{attribute 'object_name' := 'sta_TurnEmptyBusy'}
METHOD PROTECTED sta_TurnEmptyBusy : BOOL
// state implemetation
//--------------------------------------------------------------------------------------
// Entry action
	IF (me.StateMachine.intState<>me.StateMachine.intStateLastCycle) THEN
		me.StateMachine.intStateLastCycle := me.StateMachine.intState;
//		Log Message ---------------------
//		TC2_SYSTEM.ADSLOGSTR(ADSLOG_MSGTYPE_LOG,'%s','sta_TurnEmptyBusy');
//		---------------------------------
		(*p_fbMalteser^.CtrlSIf^.Par.*)intTurnDirection := E_TURN_DIRECTION.AUTOMATIC;
		(*p_fbMalteser^.CtrlSIf^.Par.*)uinPositionToGo := SIf.Cur.rInOutPosition.uinInput;
		
		IF (SIf.Cfg.bolRaxEnable) THEN
			IF SIf.Cur.rInOutPosition.uinInput*90*10 = p_fbRAX^.CtrlSIf^.Cur.dinModPosition_0_1deg THEN
				p_fbRAX^.CtrlCIf^.Job.intACmd := cCMD_STOP;
				me.SubStateMachine.intState := PTS_CmdState.cSUB_WAIT_DONE;
				me.SubStateMachine.intStateNext := PTS_CmdState.cSUB_WAIT_DONE;
			ELSE	
				p_fbRAX^.CtrlCIf^.Job.intACmd := RAX_CmdState.cCMD_TURN;
				me.SubStateMachine.intState := PTS_CmdState.cSUB_TURNbusy;
				me.SubStateMachine.intStateNext := PTS_CmdState.cSUB_TURNbusy;
			END_IF
		ELSE
			IF SIf.Cur.rInOutPosition.uinInput = p_fbMalteser^.CtrlSIf^.Cur.uintActualPosition THEN
				p_fbMalteser^.CtrlCIf^.Job.intACmd := BASE_PLC.cCMD_RUN;
				me.SubStateMachine.intState := PTS_CmdState.cSUB_WAIT_DONE;
				me.SubStateMachine.intStateNext := PTS_CmdState.cSUB_WAIT_DONE;
			ELSE	
				p_fbMalteser^.CtrlCIf^.Job.intACmd := MDC_CmdState.cCMD_TURN;
				me.SubStateMachine.intState := PTS_CmdState.cSUB_TURNbusy;
				me.SubStateMachine.intStateNext := PTS_CmdState.cSUB_TURNbusy;
			END_IF
		END_IF
	END_IF


//--------------------------------------------------------------------------------------
// Cyclic action
	IF (me.StateMachine.intState=me.StateMachine.intStateLastCycle) THEN
		//--------------------------------------------------------------------------------------
		// sub state machine for sequence
		IF (SIf.Cfg.bolRaxEnable) THEN
			CASE me.SubStateMachine.intState OF
				//--------------------------------------------------------------------------------------
				PTS_CmdState.cSUB_TURNbusy :
					IF (p_fbRAX^.CtrlCIf^.Job.intState = RAX_CmdState.cSTA_TURN) THEN
						p_fbRAX^.CtrlCIf^.Job.intACmd := cCMD_STOP;
						me.SubStateMachine.intStateNext := PTS_CmdState.cSUB_WAIT_DONE;
					END_IF
				//--------------------------------------------------------------------------------------
				PTS_CmdState.cSUB_WAIT_DONE:
					IF (p_fbRAX^.CtrlCIf^.Job.intState = cSTA_STOP) THEN
						IF SIf.Par.eMode = E_PTS_MODE.Distribute THEN
							SIf.Cur.iActualDistributionIndex := (SIf.Cur.iActualDistributionIndex + 1) MOD PTS_CmdState.cPTS_MAX_DISTRIBUTION;	
						END_IF
	
						me.StateMachine.intStateNext := BASE_PLC.cSTA_RUNBusy;
					END_IF
				//--------------------------------------------------------------------------------------
			END_CASE
		ELSE			
			CASE me.SubStateMachine.intState OF
				//--------------------------------------------------------------------------------------
				PTS_CmdState.cSUB_TURNbusy :
					IF (p_fbMalteser^.CtrlCIf^.Job.intState = MDC_CmdState.cSTA_TURNDONE) THEN
						p_fbMalteser^.CtrlCIf^.Job.intACmd := BASE_PLC.cCMD_RUN;
						me.SubStateMachine.intStateNext := PTS_CmdState.cSUB_WAIT_DONE;
					END_IF
				//--------------------------------------------------------------------------------------
				PTS_CmdState.cSUB_WAIT_DONE:
					IF (p_fbMalteser^.CtrlCIf^.Job.intState = MDC_CmdState.cSTA_InPosition) THEN
						IF SIf.Par.eMode = E_PTS_MODE.Distribute THEN
							SIf.Cur.iActualDistributionIndex := (SIf.Cur.iActualDistributionIndex + 1) MOD PTS_CmdState.cPTS_MAX_DISTRIBUTION;	
						END_IF
	
						me.StateMachine.intStateNext := BASE_PLC.cSTA_RUNBusy;
					END_IF
				//--------------------------------------------------------------------------------------
			END_CASE
		END_IF
	END_IF


//--------------------------------------------------------------------------------------
// Exit action
	IF (me.StateMachine.intState<>me.StateMachine.intStateNext) THEN
		;
	END_IF
END_METHOD

{attribute 'object_name' := 'IoOutBridge'}
METHOD PROTECTED IoOutBridge : BOOL
VAR
	bolSwitchValvesOff: BOOL;
END_VAR
// digitale and analoge inputs read from hardware or forcing
IF (CIf.SwCfg.bolSimulation = FALSE) THEN
	;
END_IF

// Write Outputs to Turning Child (Malteser or ServoDrive)
IF (SIf.Cfg.bolRaxEnable) THEN
	// ToDo: p_fbRAX^.CtrlSIf^.Par. intTurnDirection := intTurnDirection;
	p_fbRAX^.CtrlSIf^.Par.dinPos_0_1Deg := uinPositionToGo*90*10;	
ELSE
	p_fbMalteser^.CtrlSIf^.Par.intTurnDirection := intTurnDirection;	// <0 = Turn left; =0 automatic; >0 turn right
	p_fbMalteser^.CtrlSIf^.Par.uinPositionToGo := uinPositionToGo;
END_IF
END_METHOD

{attribute 'object_name' := 'sta_PON'}
METHOD PROTECTED sta_PON : BOOL
// state implemetation
//--------------------------------------------------------------------------------------
// Entry action
	IF (me.StateMachine.intState<>me.StateMachine.intStateLastCycle) THEN
		me.StateMachine.intStateLastCycle := me.StateMachine.intState;
		
	END_IF


//--------------------------------------------------------------------------------------
// Cyclic action
	IF (me.StateMachine.intState=me.StateMachine.intStateLastCycle) THEN
		;
	END_IF




//--------------------------------------------------------------------------------------
// Exit action
	IF (me.StateMachine.intState<>me.StateMachine.intStateNext) THEN
		;
	END_IF
END_METHOD

{attribute 'object_name' := 'sta_PaperDelayBusy'}
METHOD PROTECTED sta_PaperDelayBusy : BOOL
// state implemetation
//--------------------------------------------------------------------------------------
// Entry action
	IF (me.StateMachine.intState<>me.StateMachine.intStateLastCycle) THEN
		me.StateMachine.intStateLastCycle := me.StateMachine.intState;
//		Log Message ---------------------
		TC2_SYSTEM.ADSLOGSTR(ADSLOG_MSGTYPE_LOG,'%s','sta_PaperDelayBusy');
//		---------------------------------
	END_IF


//--------------------------------------------------------------------------------------
// Cyclic action
	IF (me.StateMachine.intState = me.StateMachine.intStateLastCycle) THEN
		IF (me.StateMachine.udiTimeInState_ms > SIf.Par.udiPaperInTurnDelayTime) THEN
			me.StateMachine.intStateNext := PTS_CmdState.cSTA_TurnPaperBusy;
		END_IF
	END_IF


//--------------------------------------------------------------------------------------
// Exit action
	IF (me.StateMachine.intState<>me.StateMachine.intStateNext) THEN
		;
	END_IF
END_METHOD

{attribute 'object_name' := 'sta_RUNBusy'}
METHOD PROTECTED sta_RUNBusy : BOOL
// state implemetation
//--------------------------------------------------------------------------------------
// Entry action
IF (me.StateMachine.intState<>me.StateMachine.intStateLastCycle) THEN
	me.StateMachine.intStateLastCycle := me.StateMachine.intState;

	CASE SIf.Par.eMode OF
		E_PTS_MODE.Automatic:
			pfbAlarmCtrl^.setAlarm(CIf.Info.intCtrlId,INT_TO_UINT(E_ALM_PTS.ModeParameter),0,ADR(SIf.Alm),E_AlmState.RST,CIf.Job.eMe_ActivAlmClass);
(*
			IF SIf.Cfg.bolBarcodeReaderAvailable (* AND BCR has a new barcode read *) THEN
				me.StateMachine.intStateNext := PTS_CmdState.cSTA_GetItemBusy;
			ELSE
				pfbAlarmCtrl^.setAlarm(CIf.Info.intCtrlId,INT_TO_UINT(E_ALM_PTS.ModeParameter),0,ADR(SIf.Alm),E_AlmState.RST,CIf.Job.eMe_ActivAlmClass);
			END_IF
*)
		E_PTS_MODE.Distribute:
			SIf.Cur.rInOutPosition := SIf.Cfg.aFixPosDef[SIf.Cfg.aDistributionPositionDefinition[SIf.Cur.iActualDistributionIndex]];

		ELSE
			SIf.Cur.rInOutPosition := SIf.Cfg.aFixPosDef[SIf.Par.eMode];
	END_CASE

	(*p_fbMalteser^.CtrlSIf^.Par.*)intTurnDirection := E_TURN_DIRECTION.AUTOMATIC;
	(*p_fbMalteser^.CtrlSIf^.Par.*)uinPositionToGo := SIf.Cur.rInOutPosition.uinOutput;

	IF (SIf.Cfg.bolRaxEnable = FALSE) THEN
		IF SIf.Cfg.bolPositionMalteserEnable THEN
			p_fbMalteser^.CtrlCIf^.Job.intACmd := MDC_CmdState.cCMD_PREPOSITION;
	
			me.SubStateMachine.intState := PTS_CmdState.cSUB_PREPOSITIONbusy;
			me.SubStateMachine.intStateNext := PTS_CmdState.cSUB_PREPOSITIONbusy;
		ELSE	
			p_fbMalteser^.CtrlCIf^.Job.intACmd := BASE_PLC.cCMD_RUN;
	
			me.SubStateMachine.intState := PTS_CmdState.cSUB_WAIT_DONE;
			me.SubStateMachine.intStateNext := PTS_CmdState.cSUB_WAIT_DONE;
		END_IF
	END_IF
	
	p_fbBelt^.CtrlSIf^.Par.intDirection := E_BELT_DIRECTION.FORWARD;
	pBeltCIf^.Job.intACmd := BASE_PLC.cCMD_RUN;
END_IF


//--------------------------------------------------------------------------------------
// Cyclic action
IF (me.StateMachine.intState=me.StateMachine.intStateLastCycle) THEN

	IF (SIf.Cfg.bolRaxEnable) THEN
		me.StateMachine.intStateNext := cSTA_RUN;
	ELSE
		//--------------------------------------------------------------------------------------
		// sub state machine for sequence
		CASE me.SubStateMachine.intState OF
			//--------------------------------------------------------------------------------------
			PTS_CmdState.cSUB_PREPOSITIONbusy:
				IF (p_fbMalteser^.CtrlCIf^.Job.intState = MDC_CmdState.cSTA_PREPOSITION) THEN
					p_fbMalteser^.CtrlCIf^.Job.intACmd := BASE_PLC.cCMD_RUN;
					me.SubStateMachine.intStateNext := PTS_CmdState.cSUB_WAIT_DONE;
				END_IF
			//--------------------------------------------------------------------------------------
			PTS_CmdState.cSUB_WAIT_DONE:
				IF (p_fbMalteser^.CtrlCIf^.Job.intState = MDC_CmdState.cSTA_InPosition) 
				  AND (pBeltCIf^.Job.intState = BASE_PLC.cSTA_RUN) THEN
		//			SIf.Cur.udiPaperInTurnDelayTime := 150000 / p_fbBelt^.CtrlSIf^.Par.uinBeltSpeed;
		//			SIf.Cur.udiPaperOutTurnDelayTime := CalculateOutputDelay(p_fbBelt^.CtrlSIf^.Par.uinBeltSpeed,SIf.Cur.udiPaperInTurnDelayTime);
					me.StateMachine.intStateNext := BASE_PLC.cSTA_RUN;
				END_IF
			//--------------------------------------------------------------------------------------
		END_CASE
	END_IF
	
	IF SIf.In.bolPaperAvailable.intern THEN
		me.StateMachine.intStateNext := PTS_CmdState.cSTA_WaitPaper;
	END_IF
END_IF


//--------------------------------------------------------------------------------------
// Exit action
IF (me.StateMachine.intState<>me.StateMachine.intStateNext) THEN
	;
END_IF
END_METHOD

{attribute 'object_name' := 'sta_GetItemBusy'}
METHOD PROTECTED sta_GetItemBusy : BOOL
END_METHOD

{attribute 'object_name' := 'CtrlInit'}
METHOD CtrlInit : BOOL
SUPER^.CtrlInit();

IF (SIf.Cfg.bolRaxEnable) THEN
	THIS^.AddChild(p_fbRAX^);

	pRaxCIf := p_fbRAX^.CtrlCIf;
ELSE
	THIS^.AddChild(p_fbMalteser^);

	pMalteserCIf := p_fbMalteser^.CtrlCIf;
END_IF

THIS^.AddChild(p_fbBelt^);

pBeltCIf := p_fbBelt^.CtrlCIf;

(*
// set parent id
pMalteserCIf^.Info.intParentCtrlId := CIf.Info.intCtrlId;			
pBeltCIf^.Info.intParentCtrlId := CIf.Info.intCtrlId;			

//necessary???
THIS^.CIf.Info.p_aCIf[0] := pMalteserCIf;
THIS^.CIf.Info.p_aCIf[1] := pBeltCIf;
*)
END_METHOD

{attribute 'object_name' := 'sta_ERROR'}
METHOD PROTECTED sta_ERROR : BOOL
// state implemetation
//--------------------------------------------------------------------------------------
// Entry action
	IF (me.StateMachine.intState<>me.StateMachine.intStateLastCycle) THEN
		me.StateMachine.intStateHistory := me.StateMachine.intStateLastCycle; // -> possibillity to go back to state before error
		me.StateMachine.intStateLastCycle := me.StateMachine.intState;
		
		// stop child controllers
		pBeltCIf^.Job.intACmd := BASE_PLC.cCMD_OFF;
		IF (SIf.Cfg.bolRaxEnable) THEN
			pRaxCIf^.Job.intACmd := cCMD_OFF;
		ELSE
			pMalteserCIf^.Job.intACmd := BASE_PLC.cCMD_OFF;
		END_IF
	END_IF


//--------------------------------------------------------------------------------------
// Cyclic action
	IF (me.StateMachine.intState=me.StateMachine.intStateLastCycle) THEN
		
		;
		
		
		// State Change Condition
		IF (CIf.Job.bolAlmReset = TRUE) THEN
			me.StateMachine.intStateNext := cSTA_ERRORQuit;
		END_IF
	END_IF




//--------------------------------------------------------------------------------------
// Exit action
	IF (me.StateMachine.intState<>me.StateMachine.intStateNext) THEN
		;
	END_IF
END_METHOD

{attribute 'object_name' := 'getCtrlSIf'}
METHOD getCtrlSIf : POINTER TO T_Ctrl_SIf_PTS
getCtrlSIf := ADR(SIf);
END_METHOD

END_FUNCTION_BLOCK

// ---- POUs/Controller/Lvl2/PTS [Paper Turning Station]/helper/cycle_Pts.TcPOU
FUNCTION cycle_Pts : BOOL
VAR_INPUT
	pPts: POINTER TO T_PTS;
END_VAR

pPts^.ctrl.fbPts_Ptb_Umc.In_uinStatus 				:= pPts^.io.In_uinPtb_Umc_Status;
pPts^.ctrl.fbPts_Ptb_Umc.In_intMotorActualSpeed		:= pPts^.io.In_uinPtb_Umc_ActualSpeed;
pPts^.ctrl.fbPts_Ptb_Umc.In_uinMotorSetSpeed		:= pPts^.io.In_uinPtb_Umc_SetSpeed;
pPts^.ctrl.fbPts_Ptb_Umc.In_uinIOData				:= pPts^.io.In_uinPtb_Umc_IOData1;
pPts^.ctrl.fbPts_Ptb_Umc.In_uinECATState 			:= pPts^.io.In_uinPtb_Umc_ECatState;
pPts^.ctrl.fbPts_Ptb_Umc.In_strNetId 				:= pPts^.io.In_strPtb_Umc_ECatNetId;
pPts^.ctrl.fbPts_Ptb_Umc.In_uintPort 				:= pPts^.io.In_uinPtb_Umc_ECatPort;
pPts^.ctrl.fbPts_Ptb_Umc();
pPts^.io.Out_uinPtb_Umc_SetSpeed 					:= pPts^.ctrl.fbPts_Ptb_Umc.Out_uinSpeedSetpoint;
pPts^.io.Out_uinPtb_Umc_Control 					:= pPts^.ctrl.fbPts_Ptb_Umc.Out_uinControl;

pPts^.ctrl.fbPts_Ptb_Vpc.In_bolPumpOk 				:= pPts^.io.In_bolPtb_Vpc_PumpOk;
pPts^.ctrl.fbPts_Ptb_Vpc.In_bolVacuumOk 			:= pPts^.io.In_bolPtb_Vpc_VacuumSensor;
pPts^.ctrl.fbPts_Ptb_Vpc();
pPts^.io.Out_bolPtb_Vpc_PumpOn 						:= pPts^.ctrl.fbPts_Ptb_Vpc.Out_bolVaccumPumpOn;

IF (pPts^.ctrl.fbPts.CtrlSIf^.Cfg.bolRaxEnable = FALSE) THEN
	pPts^.ctrl.fbPts_Mdc_Umc.In_uinStatus 				:= pPts^.io.In_uinMdc_Umc_Status;
	pPts^.ctrl.fbPts_Mdc_Umc.In_intMotorActualSpeed		:= pPts^.io.In_uinMdc_Umc_ActualSpeed;
	pPts^.ctrl.fbPts_Mdc_Umc.In_uinMotorSetSpeed 		:= pPts^.io.In_uinMdc_Umc_SetSpeed;
	pPts^.ctrl.fbPts_Mdc_Umc.In_uinIOData				:= pPts^.io.In_uinMdc_Umc_IOData1;
	pPts^.ctrl.fbPts_Mdc_Umc.In_uinECATState 			:= pPts^.io.In_uinMdc_Umc_ECatState;
	pPts^.ctrl.fbPts_Mdc_Umc.In_strNetId 				:= pPts^.io.In_strMdc_Umc_ECatNetId;
	pPts^.ctrl.fbPts_Mdc_Umc.In_uintPort 				:= pPts^.io.In_uinMdc_Umc_ECatPort;
	pPts^.ctrl.fbPts_Mdc_Umc();
	pPts^.io.Out_uinMdc_Umc_SetSpeed 					:= pPts^.ctrl.fbPts_Mdc_Umc.Out_uinSpeedSetpoint;
	pPts^.io.Out_uinMdc_Umc_Control 					:= pPts^.ctrl.fbPts_Mdc_Umc.Out_uinControl;
	
	pPts^.ctrl.fbPts_Mdc.In_bolCrossPositionSensor 		:= pPts^.io.In_bolMdc_CrossPositionSensor;
	pPts^.ctrl.fbPts_Mdc.In_bolTablePositionSensor 		:= pPts^.io.In_bolMdc_TablePositionSensor;
	pPts^.ctrl.fbPts_Mdc();
ELSE
	pPts^.ctrl.fbPts_RAX_POD.In_bolHomeSwitch			:= pPts^.io.In_bolRax_PositionSensor;
	pPts^.ctrl.fbPts_RAX_POD();

	pPts^.ctrl.fbPts_RAX();
END_IF

pPts^.ctrl.fbPts_Ptb();

pPts^.ctrl.fbPts.In_bol_PaperAvailable 				:= pPts^.io.In_bolPaperSensor;
pPts^.ctrl.fbPts();

END_FUNCTION

// ---- POUs/Controller/Lvl2/PTS [Paper Turning Station]/helper/init_Pts.TcPOU
FUNCTION init_Pts : BOOL
VAR_INPUT
	pPts			: POINTER TO T_PTS;
	/// instance array of all controller instances
	pCtrlInst		: POINTER TO fb_CtrlBase;
	/// common interface array of all controllers (main use for PLC)
	pCtrlCIf		: POINTER TO T_Ctrl_CIf;
END_VAR

pPts^.ctrl.fbPts_Ptb_Vpc.iniAllCtrlArrays(pCtrlInst,pCtrlCIf,pPts^.id.Pts_Ptb_Vpc);
pPts^.ctrl.fbPts_Ptb_Umc.iniAllCtrlArrays(pCtrlInst,pCtrlCIf,pPts^.id.Pts_Ptb_Umc);
pPts^.ctrl.fbPts_Ptb.iniAllCtrlArrays(pCtrlInst,pCtrlCIf,pPts^.id.Pts_Ptb);
pPts^.ctrl.fbPts_Ptb.Drive := ADR(pPts^.ctrl.fbPts_Ptb_Umc);
pPts^.ctrl.fbPts_Ptb.VacuumPump := ADR(pPts^.ctrl.fbPts_Ptb_Vpc);

pPts^.ctrl.fbPts_Mdc_Umc.iniAllCtrlArrays(pCtrlInst,pCtrlCIf,pPts^.id.Pts_Mdc_Umc);
pPts^.ctrl.fbPts_Mdc.iniAllCtrlArrays(pCtrlInst,pCtrlCIf,pPts^.id.Pts_Mdc);
pPts^.ctrl.fbPts_Mdc.Drive := ADR(pPts^.ctrl.fbPts_Mdc_Umc);

pPts^.ctrl.fbPts_RAX.iniAllCtrlArrays(pCtrlInst,pCtrlCIf,pPts^.id.Pts_RAX);
pPts^.ctrl.fbPts_RAX.In_pAD_SIf:= pPts^.ctrl.fbPts_RAX_POD.AD_SIf;	

pPts^.ctrl.fbPts.iniAllCtrlArrays(pCtrlInst,pCtrlCIf,pPts^.id.Pts);
pPts^.ctrl.fbPts.Belt := ADR(pPts^.ctrl.fbPts_Ptb);
pPts^.ctrl.fbPts.Malteser := ADR(pPts^.ctrl.fbPts_Mdc);
pPts^.ctrl.fbPts.Servo := ADR(pPts^.ctrl.fbPts_RAX);

END_FUNCTION

// ---- POUs/Controller/Utility/Data Channel/OvenMessage/FB_OvenSendDch.TcPOU
FUNCTION_BLOCK FB_OvenSendDch EXTENDS FB_DataChannelSendBase IMPLEMENTS I_DataChannelSend
VAR
	/// Saber Inteface Variables
	/// -----------------------------------------------------------------
	m_pOutputData: POINTER TO T_Oven_DCH;
END_VAR

(* Copyright 2017 Cimpress

Licensed under the Apache License, Version 2.0 (the "License");
you may not use this file except in compliance with the License.
You may obtain a copy of the License at

http://www.apache.org/licenses/LICENSE-2.0

Unless required by applicable law or agreed to in writing, software
distributed under the License is distributed on an "AS IS" BASIS,
WITHOUT WARRANTIES OR CONDITIONS OF ANY KIND, either express or implied.
See the License for the specific language governing permissions and
limitations under the License. *)

SUPER^();

{attribute 'object_name' := 'SendData'}
METHOD SendData : BOOL
VAR_INPUT
	udiDataSize: UDINT;
	pData: POINTER TO BYTE;
END_VAR
SendData := FALSE;

IF m_eState = E_PlcSaberDHCState.WaitForJob THEN
	IF (udiDataSize > 0 ) AND (pData <> TC3_MEMMAN.NULL) THEN
		TC2_SYSTEM.MEMCPY(destAddr := m_pOutputData, srcAddr := pData, n := udiDataSize);
		m_eState := E_PlcSaberDHCState.SendData;	
		SendData := TRUE;
	END_IF	
END_IF
END_METHOD

{attribute 'object_name' := 'InitChannel'}
METHOD InitChannel : BOOL
VAR_INPUT
	udiDataSize: UDINT;
	pOutputData: POINTER TO BYTE;
END_VAR
InitChannel := FALSE;

IF udiDataSize > 0 THEN
	IF pOutputData <> TC3_MEMMAN.NULL THEN
		m_uinDataSize := udiDataSize;
		m_pOutputData := pOutputData;
		m_eState := E_PlcSaberDHCState.Init;
		InitChannel := TRUE;
	END_IF
END_IF
END_METHOD

END_FUNCTION_BLOCK

// ---- POUs/Controller/Utility/Data Channel/PrintDoneMessage/FB_JCL_PrintDoneSendDch.TcPOU
FUNCTION_BLOCK FB_JCL_PrintDoneSendDch EXTENDS FB_DataChannelSendBase IMPLEMENTS I_DataChannelSend
VAR
	/// Saber Inteface Variables
	/// -----------------------------------------------------------------
	m_pOutputData: POINTER TO T_JCL_DCH;
END_VAR

(* Copyright 2017 Cimpress

Licensed under the Apache License, Version 2.0 (the "License");
you may not use this file except in compliance with the License.
You may obtain a copy of the License at

http://www.apache.org/licenses/LICENSE-2.0

Unless required by applicable law or agreed to in writing, software
distributed under the License is distributed on an "AS IS" BASIS,
WITHOUT WARRANTIES OR CONDITIONS OF ANY KIND, either express or implied.
See the License for the specific language governing permissions and
limitations under the License. *)

SUPER^();

{attribute 'object_name' := 'SendData'}
METHOD SendData : BOOL
VAR_INPUT
	udiDataSize: UDINT;
	pData: POINTER TO BYTE;
END_VAR
SendData := FALSE;

IF m_eState = E_PlcSaberDHCState.WaitForJob THEN
	IF (udiDataSize > 0 ) AND (pData <> TC3_MEMMAN.NULL) THEN
		TC2_SYSTEM.MEMCPY(destAddr := m_pOutputData, srcAddr := pData, n := udiDataSize);
		m_eState := E_PlcSaberDHCState.SendData;	
		SendData := TRUE;
	END_IF	
END_IF
END_METHOD

{attribute 'object_name' := 'InitChannel'}
METHOD InitChannel : BOOL
VAR_INPUT
	udiDataSize: UDINT;
	pOutputData: POINTER TO BYTE;
END_VAR
InitChannel := FALSE;

IF udiDataSize > 0 THEN
	IF pOutputData <> TC3_MEMMAN.NULL THEN
		m_uinDataSize := udiDataSize;
		m_pOutputData := pOutputData;
		m_eState := E_PlcSaberDHCState.Init;
		InitChannel := TRUE;
	END_IF
END_IF
END_METHOD

END_FUNCTION_BLOCK

// ---- POUs/Controller/Utility/FiFo/FB_DataSetFifo.TcPOU
FUNCTION_BLOCK FB_DataSetFifo
VAR_INPUT
	bOverwrite: BOOL;
	in: POINTER TO BYTE;
	iAddSize: INT;
END_VAR
VAR_OUTPUT
	bOk: BOOL;
	nCount: UDINT;
	nLoad: UDINT;
	out: ARRAY[0..MAX_DATASET_SIZE] OF BYTE;
	pHeader: POINTER TO ST_Header;
END_VAR
VAR
	/// Buffer memory used by FB_MemRingBuffer function block 
	arrBuffer: ARRAY[0..MAX_BUFFER_SIZE] OF BYTE;
	fbBuffer: FB_MemRingBuffer;
	intLoopRemove: INT;
	intLoopReset: INT;
END_VAR
VAR CONSTANT
	MAX_BUFFER_SIZE: UDINT := 1000;
END_VAR

;

ACTION A_Add:
fbBuffer.A_AddTail( pWrite:= in,
					cbWrite:= INT_TO_UDINT(iAddSize),
					pBuffer:= ADR( arrBuffer ),
					cbBuffer:= SIZEOF( arrBuffer ),
					bOk=> bOk,
					nCount => nCount );

IF NOT bOk THEN (* overflow ? *)
	IF bOverwrite THEN
		fbBuffer.A_RemoveHead(); (* remove one oldest entry *)
		fbBuffer.A_AddTail( bOk => bOk, nCount => nCount );
	END_IF
END_IF

nLoad := (fbBuffer.cbSize * 100) / MAX_BUFFER_SIZE;
END_ACTION

ACTION A_Get:
fbBuffer.A_GetHead( pRead:= ADR( out ),
					cbRead:= SIZEOF( out ),
					pBuffer:= ADR( arrBuffer ),
					cbBuffer:= SIZEOF( arrBuffer ),
					bOk=> bOk,
					nCount => nCount );

pHeader := ADR(out);					
					
nLoad := (fbBuffer.cbSize * 100) / MAX_BUFFER_SIZE;
END_ACTION

ACTION A_Reset:
// MEMSET not working!
//MEMSET( ADR( arrBuffer ), 0, SIZEOF( arrBuffer ) ); (* reset (optional) internal buffer *)
FOR intLoopReset:=0 TO SIZEOF(arrBuffer)-1 DO
	arrBuffer[intLoopReset]:= 0;
END_FOR

fbBuffer.A_Reset( 	bOk=> bOk,
					nCount => nCount );

nLoad := (fbBuffer.cbSize * 100) / MAX_BUFFER_SIZE;
END_ACTION

ACTION A_Remove:
// Clean up package buffer
FOR intLoopRemove:=0 TO SIZEOF(out)-1 DO
	out[intLoopRemove]:= 0;
END_FOR

// Remove data from buffer. Get next package.
fbBuffer.A_RemoveHead( 	pRead:= ADR(out),
						cbRead:= SIZEOF(out),
						pBuffer:= ADR(arrBuffer),
						cbBuffer:= SIZEOF(arrBuffer),
						bOk=> bOk,
						nCount => nCount );
// Return						
pHeader := ADR(out);

nLoad := (fbBuffer.cbSize * 100) / MAX_BUFFER_SIZE;
END_ACTION

END_FUNCTION_BLOCK

// ---- POUs/Controller/Utility/LookupTable/FB_LookupTable.TcPOU
FUNCTION_BLOCK FB_LookupTable
VAR_INPUT
	iAddKey: INT;
	iAddValue: INT;
	iLookupKey: INT;
	iLookupValue: INT;
END_VAR
VAR_OUTPUT
	/// number of elements in Table
	iCount: INT;
	bOK: BOOL;
	iFoundValue: INT;
	iFoundKey: INT;
END_VAR
VAR
	aiKeys: ARRAY[0..MaxLookupSize] OF INT;
	aiValues: ARRAY[0..MaxLookupSize] OF INT;
	ii: INT;
	bDone: BOOL;
END_VAR

(* 
	This is a very slow lookup table! do not use for big amounts of data
*)

ACTION A_Add:
IF (iAddKey = 0) OR (iCount = MaxLookupSize) THEN
	bOK := 0; 
	RETURN;
END_IF
bDone := 0;

FOR ii := 0 TO MaxLookupSize BY 1 DO // see if key already exists
	IF ( iAddKey = aiKeys[ii] ) THEN // overwrite old element
		aiValues[ii] := iAddValue;
		bOK := 1;
		bDone := 1;
		RETURN;
	END_IF
END_FOR

// add new entry
// find first unused element in table
FOR ii := 0 TO MaxLookupSize BY 1 DO
	IF aiKeys[ii] = 0 THEN
		aiKeys[ii] := iAddKey;
		aiValues[ii] := iAddValue;
		iCount := iCount +1;
		bOK := 1;
		RETURN;
	END_IF
END_FOR
END_ACTION

ACTION A_Reset:
FOR ii := 0 TO MaxLookupSize BY 1 DO
	aiKeys[ii] := 0;
	aiValues[ii] := 0;
END_FOR
bOK := 1;
END_ACTION

ACTION A_RemoveKey:
bOK := 0;

FOR ii := 0 TO MaxLookupSize BY 1 DO
	IF iLookupKey = aiKeys[ii] THEN // found it
		aiKeys[ii] := 0;
		aiValues[ii] := 0;
		bOK := 1;
		RETURN;
	END_IF
END_FOR
END_ACTION

ACTION A_LookupByValue:
// will only find the first key associated with the value
bOK := 0;

FOR ii := 0 TO MaxLookupSize BY 1 DO
	IF iLookupValue = aiValues[ii] THEN // found it
		iFoundKey := aiKeys[ii];
		bOK := 1;
		RETURN;
	END_IF
END_FOR
END_ACTION

ACTION A_LookupByKey:
bOK := 0;

FOR ii := 0 TO MaxLookupSize BY 1 DO
	IF iLookupKey = aiKeys[ii] THEN // found it
		iFoundValue := aiValues[ii];
		bOK := 1;
		RETURN;
	END_IF
END_FOR
END_ACTION

END_FUNCTION_BLOCK

// ---- POUs/Controller/Utility/LookupTable/FB_LookupTable_String.TcPOU
FUNCTION_BLOCK FB_LookupTable_String
VAR_INPUT
	iAddKey: INT;
	strAddValue: STRING;
	iLookupKey: INT;
	strLookupValue: STRING;
END_VAR
VAR_OUTPUT
	/// number of elements in Table
	iCount: INT;
	bOK: BOOL;
	strFoundValue: STRING;
	iFoundKey: INT;
END_VAR
VAR
	_aiKeys: ARRAY[0..MaxLookupSize] OF INT;
	_astrValues: ARRAY[0..MaxLookupSize] OF STRING;
	_iIdx: INT;
	_bDone: BOOL;
END_VAR

(* 
	This is a very slow lookup table! do not use for big amounts of data
*)

ACTION A_Add:
IF (iAddKey = 0) OR (iCount = MaxLookupSize) THEN
	bOK := 0; 
	RETURN;
END_IF
_bDone := 0;

FOR _iIdx := 0 TO MaxLookupSize BY 1 DO // see if key already exists
	IF ( iAddKey = _aiKeys[_iIdx] ) THEN // overwrite old element
		_astrValues[_iIdx] := strAddValue;
		bOK := 1;
		_bDone := 1;
		RETURN;
	END_IF
END_FOR

// add new entry
// find first unused element in table
FOR _iIdx := 0 TO MaxLookupSize BY 1 DO
	IF _aiKeys[_iIdx] = 0 THEN
		_aiKeys[_iIdx] := iAddKey;
		_astrValues[_iIdx] := strAddValue;
		iCount := iCount +1;
		bOK := 1;
		RETURN;
	END_IF
END_FOR
END_ACTION

ACTION A_Reset:
FOR _iIdx := 0 TO MaxLookupSize BY 1 DO
	_aiKeys[_iIdx] := 0;
	_astrValues[_iIdx] := '';
END_FOR
bOK := 1;
END_ACTION

ACTION A_RemoveKey:
bOK := 0;

FOR _iIdx := 0 TO MaxLookupSize BY 1 DO
	IF iLookupKey = _aiKeys[_iIdx] THEN // found it
		_aiKeys[_iIdx] := 0;
		_astrValues[_iIdx] := '';
		bOK := 1;
		RETURN;
	END_IF
END_FOR
END_ACTION

ACTION A_LookupByKey:
bOK := 0;

FOR _iIdx := 0 TO MaxLookupSize BY 1 DO
	IF iLookupKey = _aiKeys[_iIdx] THEN // found it
		strFoundValue := _astrValues[_iIdx];
		bOK := 1;
		RETURN;
	END_IF
END_FOR
END_ACTION

ACTION A_LookupByValue:
// will only find the first key associated with the value
bOK := 0;

FOR _iIdx := 0 TO MaxLookupSize BY 1 DO
	IF strLookupValue = _astrValues[_iIdx] THEN // found it
		iFoundKey := _aiKeys[_iIdx];
		bOK := 1;
		RETURN;
	END_IF
END_FOR
END_ACTION

END_FUNCTION_BLOCK
